FUNCTION button : BOOL
VAR_INPUT
END_VAR
VAR
END_VAR

END_FUNCTION

(* stored: Version 1.1.0.1, ProductVersion 3.1.4024.12
   POU button: Id {980a9b75-0e1f-4e75-a249-8ef7030a659a}, SpecialFunc None *)
